FUNCTION_BLOCK FB_Add2Ints
VAR_INPUT
	Int1	: INT;
	Int2	: INT;
END_VAR
VAR_OUTPUT
	Result	: INT;
END_VAR
VAR
END_VAR

END_FUNCTION_BLOCK

(* stored: Version 1.1.0.1, ProductVersion 3.1.4024.12
   POU FB_Add2Ints: Id {0818456f-bc7e-466e-9037-ec10ae069589}, SpecialFunc None *)
